# EPICS substitutions: ek9000App/Db/EL3112.substitutions
file EL3112.template
{       pattern
        {
                TERMINAL,

        }
        {
        }
}
